Staubli VAL3: goTo.pgx

program goTo(bool& x_bUnreached[], InstrItem x_iInstrItem)
  local bool l_bUnreached
  local num l_nIndexTool
  local tool l_tTool
  local num l_nSize
  local string l_sItems[2]
  local num l_nId
  local num l_nResult
  local TrajectoryItem l_tTraj
  local string l_sPath
  local num l_nIndex
begin
//  // check the cycle status
//  if !cycleStatus:bCycle and !cycleStatus:bSimulation
//    // check the working Mode
//    if cycleStatus:nWorkingMode==1 and isPowered()
//      // set the memory for the moveHold button
//      if cycleStatus:nWorkingStatus==6
//        bMoveRelease=true
//      endIf
//      // check for the index
//      if nOldIndex!=l_nIndex or (cycleStatus:nWorkingStatus!=0 and cycleStatus:nWorkingStatus!=6)
//        if !isEmpty()
//          resetMotion()
//        endIf
//        if nOldIndex!=l_nIndex
//          nOldIndex=l_nIndex
//        endIf
//      else
//        if isEmpty() and cycleStatus:nWorkingStatus==0 and bMoveRelease
//          bMoveRelease=false
//          cls()
//          // copy the item to the trajectory
//          l_sItems=x_iInstrItem.sData
//          // take the elements
//          call saveData:getPathInstr(x_iInstrItem.sType,l_sPath)
//          if l_sPath!=sPath
//            sPath=l_sPath
//            TrajItem:libLoad(l_sPath)
//          endIf
//          call TrajItem:load(l_sItems,l_nResult)
//          call TrajItem:getSizeItem(false,l_nSize)
//          // MOVE
//          do
//            if l_nIndex>0
//              call use:typeMenu(7,"<<")
//            else
//              call use:typeMenu(7,"    ")
//            endIf
//            if l_nIndex<=l_nSize
//              call use:typeMenu(8,">>")
//            else
//              call use:typeMenu(8,"    ")
//            endIf
//            // get the data to move
//            call TrajItem:getTool(l_nIndexTool)
//            call tcp:getTool(l_tTool,l_nIndexTool)
//            call TrajItem:getTrajItem(l_tTraj,l_nIndex)
//            //
//            // use a sTemp mdesc to set the blend off
//            //
//            l_tTraj.nom_speed.blend=off
//            call TrajItem:goTo(l_tTool,l_tTraj.nom_speed,l_tTraj.moveType,x_bUnreached,l_nIndex)
//            // TO DO language
//            call use:timerDialog("Going to point: "+toString("",l_nIndex+1)+ " / "+toString("",l_nSize),0)
//            do
//              l_nId=getKey()
//              call use:scroll(0,7,38,(getMoveId()-roundDown(getMoveId()))*100)
//              delay(0)
//            until isEmpty()or l_nId==255 or l_nId==277 or l_nId==278
//            // continue
//            if isEmpty() or (l_nId==278 and l_nIndex<l_nSize)
//              if isEmpty()
//                call use:timerDialog("At point: "+toString("",l_nIndex+1)+ " / "+toString("",l_nSize),1)
//              endIf
//              l_nIndex=l_nIndex+1
//            elseIf l_nId==277 and l_nIndex>0
//              // decrease
//              l_nIndex=l_nIndex-1
//            else
//              delay(1)
//            endIf
//            // release
//            resetMotion()
//          until x_bUnreached or l_nId==255 or l_nIndex>=l_nSize or(l_nIndex==l_nSize and l_nSize==1)
//          // refresh
//          use:bUseRefresh=true
//        endIf
//      endIf
//    else
//      // reset the cycle
//      if cycleStatus:nWorkingMode!=1 or !isPowered()
//        resetMotion()
//      endIf
//    endIf
//  endIf
//  if l_nId==255
//    // release
//    call use:nullKey(l_nId)
//  endIf
end
